(* PLC project Unnamed, Unknown Unnamed 1 *)
(* stored: creationDateTime 2024-09-17T16:35:19, modificationDateTime 2024-10-07T20:39:50 *)

PROGRAM program0

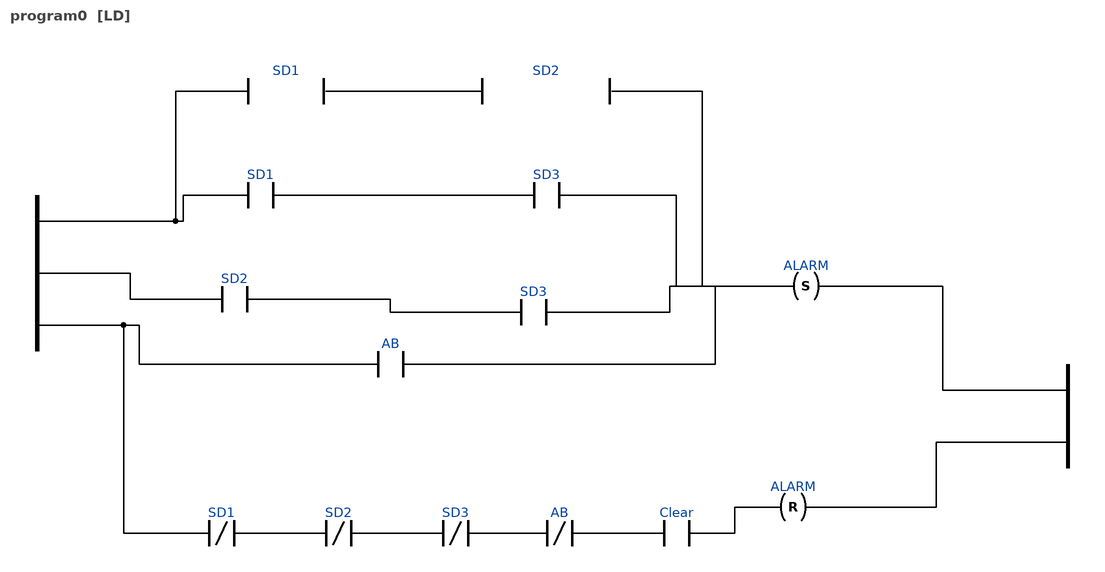
(* LD diagram, written out as Structured Text *)
IF SD1 AND SD2 OR SD1 AND SD3 OR SD2 AND SD3 OR AB THEN ALARM := TRUE; END_IF;
IF NOT SD1 AND NOT SD2 AND NOT SD3 AND NOT AB AND Clear THEN ALARM := FALSE; END_IF;
END_PROGRAM

FUNCTION function0 : BOOL

(* LD diagram, written out as Structured Text *)
END_FUNCTION

FUNCTION_BLOCK FunctionBlockDiagram1
  VAR_INPUT
    Switch1 : BOOL;
    PushBtn : BOOL;
  END_VAR
  VAR_OUTPUT
    LampGreen : BOOL;
    LampRed : BOOL;
    LampYellow : BOOL;
  END_VAR

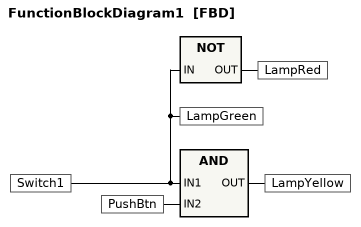
(* FBD diagram, written out as Structured Text *)
LampGreen := Switch1;
LampRed := NOT Switch1;
LampYellow := Switch1 AND PushBtn;
END_FUNCTION_BLOCK

FUNCTION_BLOCK functionBlock0
  VAR
    TON_Timer1 : TON;
    TOF_Timer2 : TOF;
  END_VAR

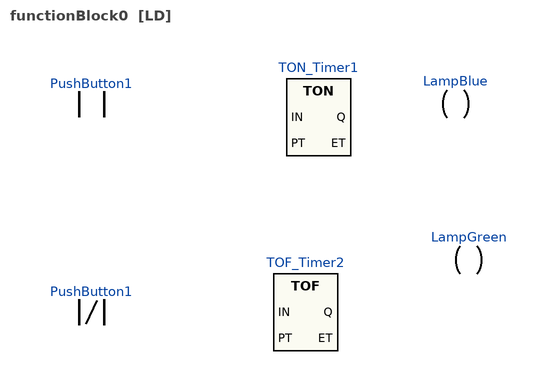
(* LD diagram, written out as Structured Text *)
TON_Timer1();
TOF_Timer2();
(* drawn but not wired to any output: PushButton1, PushButton1 *)
END_FUNCTION_BLOCK

CONFIGURATION Config0
  RESOURCE Res0 ON PLC
  END_RESOURCE
END_CONFIGURATION
